// TIA Portal V19 export
TYPE "C403_VAR_IF_LVE_TYPIC"
   STRUCT
      EXT_HW { ExternalAccessible := 'False'; ExternalVisible := 'False'; ExternalWritable := 'False'} : Bool;   // Sturings hardware (PLC) in storing
      STS_KST_OPEN { ExternalAccessible := 'False'; ExternalVisible := 'False'; ExternalWritable := 'False'} : Bool;   // TRUE = deur wegkantkast geopend
      STS_NEG { ExternalAccessible := 'False'; ExternalVisible := 'False'; ExternalWritable := 'False'} : Bool;   // Spookrijder gedetecteerd
      STS_SOS { ExternalAccessible := 'False'; ExternalVisible := 'False'; ExternalWritable := 'False'} : Bool;   // Snelheidsonderschrijding
      STS_STOP { ExternalAccessible := 'False'; ExternalVisible := 'False'; ExternalWritable := 'False'} : Bool;   // Stilstand
      STO { ExternalAccessible := 'False'; ExternalVisible := 'False'; ExternalWritable := 'False'} : Struct   // Opsomming van alle storingen
         A001 : Bool;   // Beveiliging aangesproken
         A002 : Bool;   // Storing detectiepunt
         A003 : Bool;   // Beveiliging klimaatregeling wegkantkast aangesproken
         A004 : Bool;   // Overspanningsbeveiliging aangesproken
      END_STRUCT;
   END_STRUCT;
END_TYPE
